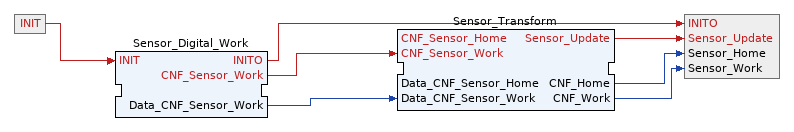
        SUBAPPLICATION Sensor_Digital_Work
          EVENT_INPUT
            INIT;
          END_EVENT
          EVENT_OUTPUT
            INITO;
            CNF_Sensor_Work;
          END_EVENT
          VAR_OUTPUT
            Data_CNF_Sensor_Work : BOOL;
          END_VAR
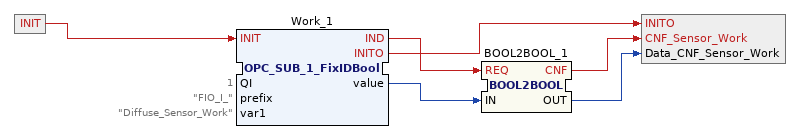
          FBS
            BOOL2BOOL_1 : BOOL2BOOL;
          END_FBS
          SUBAPPS
            Work_1 : OPC_SUB_1_FixIDBool(QI := 1, prefix := "FIO_I_", var1 := "Diffuse_Sensor_Work");
          END_SUBAPPS
          EVENT_CONNECTIONS
            Work_1.IND TO BOOL2BOOL_1.REQ;
            INIT TO Work_1.INIT;
            Work_1.INITO TO INITO;
            BOOL2BOOL_1.CNF TO CNF_Sensor_Work;
          END_CONNECTIONS
          DATA_CONNECTIONS
            Work_1.value TO BOOL2BOOL_1.IN;
            BOOL2BOOL_1.OUT TO Data_CNF_Sensor_Work;
          END_CONNECTIONS
        END_SUBAPPLICATION
        SUBAPPLICATION Sensor_Transform
          EVENT_INPUT
            CNF_Sensor_Home;
            CNF_Sensor_Work;
          END_EVENT
          EVENT_OUTPUT
            Sensor_Update;
          END_EVENT
          VAR_INPUT
            Data_CNF_Sensor_Home : BOOL;
            Data_CNF_Sensor_Work : BOOL;
          END_VAR
          VAR_OUTPUT
            CNF_Home : BOOL;
            CNF_Work : BOOL;
          END_VAR
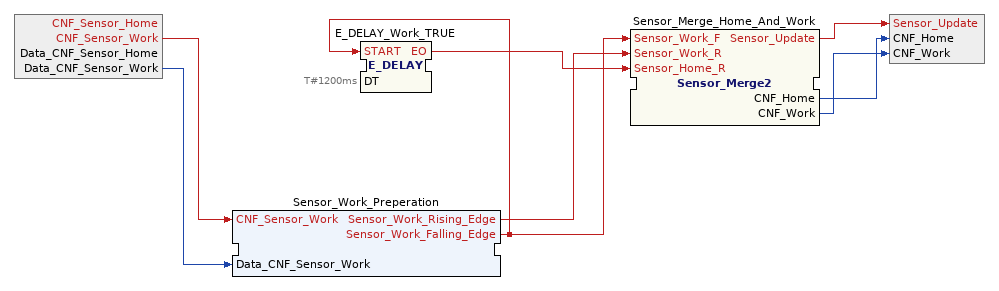
          FBS
            Sensor_Merge_Home_And_Work : Sensor_Merge2;
            E_DELAY_Work_TRUE : E_DELAY(DT := T#1200ms); (* This block mimics the function of Sensor Work. *)
          END_FBS
          SUBAPPLICATION Sensor_Work_Preperation
            EVENT_INPUT
              CNF_Sensor_Work;
            END_EVENT
            EVENT_OUTPUT
              Sensor_Work_Rising_Edge;
              Sensor_Work_Falling_Edge;
            END_EVENT
            VAR_INPUT
              Data_CNF_Sensor_Work : BOOL;
            END_VAR
            FBS
              E_F_TRIG_Work : E_F_TRIG;
              E_R_TRIG_Work : E_R_TRIG;
            END_FBS
            EVENT_CONNECTIONS
              E_F_TRIG_Work.EO TO Sensor_Work_Falling_Edge;
              E_R_TRIG_Work.EO TO Sensor_Work_Rising_Edge;
              CNF_Sensor_Work TO E_R_TRIG_Work.EI;
              CNF_Sensor_Work TO E_F_TRIG_Work.EI;
            END_CONNECTIONS
            DATA_CONNECTIONS
              Data_CNF_Sensor_Work TO E_R_TRIG_Work.QI;
              Data_CNF_Sensor_Work TO E_F_TRIG_Work.QI;
            END_CONNECTIONS
          END_SUBAPPLICATION
          EVENT_CONNECTIONS
            Sensor_Merge_Home_And_Work.Sensor_Update TO Sensor_Update;
            Sensor_Work_Preperation.Sensor_Work_Falling_Edge TO Sensor_Merge_Home_And_Work.Sensor_Work_F;
            Sensor_Work_Preperation.Sensor_Work_Rising_Edge TO Sensor_Merge_Home_And_Work.Sensor_Work_R;
            CNF_Sensor_Work TO Sensor_Work_Preperation.CNF_Sensor_Work;
            E_DELAY_Work_TRUE.EO TO Sensor_Merge_Home_And_Work.Sensor_Home_R;
            Sensor_Work_Preperation.Sensor_Work_Falling_Edge TO E_DELAY_Work_TRUE.START;
          END_CONNECTIONS
          DATA_CONNECTIONS
            Sensor_Merge_Home_And_Work.CNF_Home TO CNF_Home;
            Sensor_Merge_Home_And_Work.CNF_Work TO CNF_Work;
            Data_CNF_Sensor_Work TO Sensor_Work_Preperation.Data_CNF_Sensor_Work;
          END_CONNECTIONS
        END_SUBAPPLICATION
        EVENT_CONNECTIONS
          INIT TO Sensor_Digital_Work.INIT;
          Sensor_Digital_Work.INITO TO INITO;
          Sensor_Digital_Work.CNF_Sensor_Work TO Sensor_Transform.CNF_Sensor_Work;
          Sensor_Transform.Sensor_Update TO Sensor_Update;
        END_CONNECTIONS
        DATA_CONNECTIONS
          Sensor_Digital_Work.Data_CNF_Sensor_Work TO Sensor_Transform.Data_CNF_Sensor_Work;
          Sensor_Transform.CNF_Home TO Sensor_Home;
          Sensor_Transform.CNF_Work TO Sensor_Work;
        END_CONNECTIONS
      END_SUBAPPLICATION
      EVENT_CONNECTIONS
        HW_Control.REQ_Actuator TO Actuator.CNF_Actuator;
        HW_Control.REQ_Actuator TO Error_Control.REQ_Actuator;
        HW_Control.Moved TO Error_Control.CNF_Moved;
        Sensor.Sensor_Update TO Error_Control.Sensor_Update;
        Sensor.Sensor_Update TO HW_Control.Sensor_Update;
        Actuator.INITO TO Sensor.INIT;
        REQ_Move TO HW_Control.REQ_Move;
        HW_Control.Moved TO Moved;
        Error_Control.Error TO Error;
        INIT TO Actuator.INIT;
      END_CONNECTIONS
      DATA_CONNECTIONS
        HW_Control.Data_Actuator TO Actuator.Data_Actuator;
        Sensor.Sensor_Home TO HW_Control.Sensor_Home;
        Sensor.Sensor_Work TO HW_Control.Sensor_Work;
        Move_Destination TO HW_Control.Move_Destination;
        Error_Control.Error_Code TO Error_Code;
      END_CONNECTIONS
    END_SUBAPPLICATION
    EVENT_CONNECTIONS
      Move_Request.REQ_Move TO Hardware_Move_X.REQ_Move;
      INIT_FIO.INITO TO Hardware_Move_X.INIT;
      Hardware_Move_X.Moved TO Hardware_Move_Z.REQ_Move;
      INIT_FIO.INITO TO Hardware_Move_Z.INIT;
      INIT_FIO.INITO TO VacuumGripper.INIT;
    END_CONNECTIONS
    DATA_CONNECTIONS
      Move_Request.Move_Destination TO Hardware_Move_X.Move_Destination;
      Move_Request.Move_Destination TO Hardware_Move_Z.Move_Destination;
    END_CONNECTIONS
  END_APPLICATION
  DEVICE FORTE_PC : FORTE_PC(MGR_ID := "localhost:61499")
    {SET_ATTRIBUTE(Profile, HOLOBLOC)}
    RESOURCE EMB_RES : EMB_RES
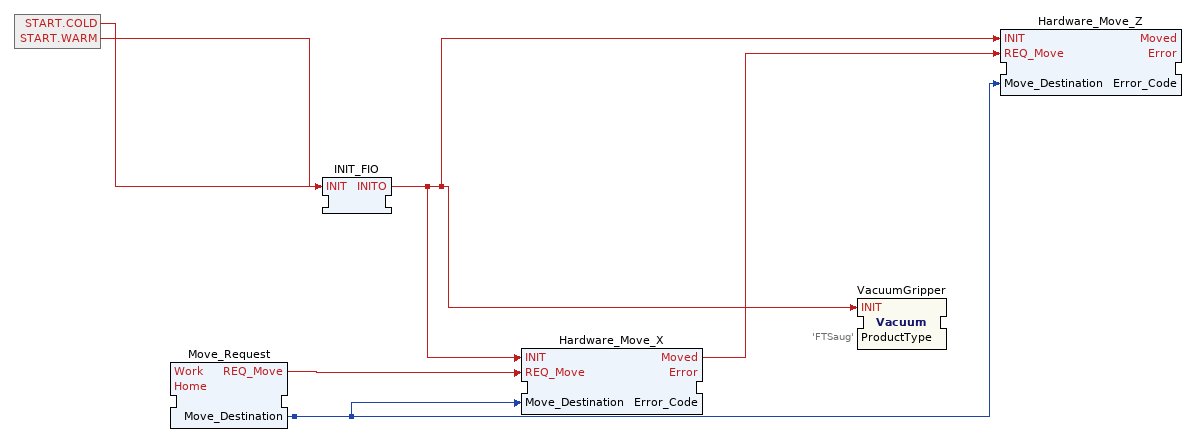
      FBS
        VacuumGripper : Vacuum(ProductType := 'FTSaug');
      END_FBS
      SUBAPPLICATION INIT_FIO
        EVENT_INPUT
          INIT;
        END_EVENT
        EVENT_OUTPUT
          INITO;
        END_EVENT
      END_SUBAPPLICATION
      SUBAPPLICATION Move_Request
        EVENT_INPUT
          Work;
          Home;
        END_EVENT
        EVENT_OUTPUT
          REQ_Move;
        END_EVENT
        VAR_OUTPUT
          Move_Destination : STRING;
        END_VAR
      END_SUBAPPLICATION
      SUBAPPLICATION Hardware_Move_X
        EVENT_INPUT
          INIT;
          REQ_Move;
        END_EVENT
        EVENT_OUTPUT
          Moved;
          Error;
        END_EVENT
        VAR_INPUT
          Move_Destination : STRING;
        END_VAR
        VAR_OUTPUT
          Error_Code : INT;
        END_VAR
      END_SUBAPPLICATION
      SUBAPPLICATION Hardware_Move_Z
        EVENT_INPUT
          INIT;
          REQ_Move;
        END_EVENT
        EVENT_OUTPUT
          Moved;
          Error;
        END_EVENT
        VAR_INPUT
          Move_Destination : STRING;
        END_VAR
        VAR_OUTPUT
          Error_Code : INT;
        END_VAR
      END_SUBAPPLICATION
      EVENT_CONNECTIONS
        START.COLD TO INIT_FIO.INIT;
        START.WARM TO INIT_FIO.INIT;
        Move_Request.REQ_Move TO Hardware_Move_X.REQ_Move;
        INIT_FIO.INITO TO Hardware_Move_X.INIT;
        Hardware_Move_X.Moved TO Hardware_Move_Z.REQ_Move;
        INIT_FIO.INITO TO Hardware_Move_Z.INIT;
        INIT_FIO.INITO TO VacuumGripper.INIT;
      END_CONNECTIONS
      DATA_CONNECTIONS
        Move_Request.Move_Destination TO Hardware_Move_X.Move_Destination;
        Move_Request.Move_Destination TO Hardware_Move_Z.Move_Destination;
      END_CONNECTIONS
    END_RESOURCE
  END_DEVICE
  MAPPINGS
    ETFA2023App.INIT_FIO ON FORTE_PC.EMB_RES.INIT_FIO;
    ETFA2023App.Move_Request ON FORTE_PC.EMB_RES.Move_Request;
    ETFA2023App.Hardware_Move_X ON FORTE_PC.EMB_RES.Hardware_Move_X;
    ETFA2023App.Hardware_Move_Z ON FORTE_PC.EMB_RES.Hardware_Move_Z;
    ETFA2023App.VacuumGripper ON FORTE_PC.EMB_RES.VacuumGripper;
  END_MAPPINGS
END_SYSTEM
